// TIA Portal V20 export
TYPE "typeEm5Standard"
// stored: Access Published, Namespace Unit1
   STRUCT
      commands { ExternalWritable := 'False'} : "Unit1.typeEm5Commands";
      monitoring { ExternalWritable := 'False'} : "Unit1.typeEm5Monitoring";
   END_STRUCT;
END_TYPE
